_CFC_ (* Continuous Function Chart, elements in execution order *)
#0 OR(SCHU_P2_4_Z_M1_AV, NOT SCHU_P2_4_SA1_DI5_A)
#1 RT_Pusk:R_TRIG(CLK: SCHU_P2_4_UST_RE_PUSK)
#2 TON_PCH_OTKL:TON(IN: SCHU_P2_4_UST_RE_STOP, PT: T#1s)
#3 FT_PCH_OTKL:R_TRIG(CLK: #2.Q)
#4 RS_YA1_Open:RS(SET: #1.Q, RESET1: #3.Q)
#5 ZADERJ_SHOD_YA1:TON(IN: #4.Q1, PT: t#10s)
#6 TON_YA1_Z_ZAM_TE2:TON(IN: SCHU_P2_4_TE2_M_ZASCH, PT: t#5s)
#7 AND(#0, #21)
#8 AND(NOT SCHU_P2_4_SA1_DI5_A, NOT SCHU_P2_4_SA8_DI3_A, NOT SCHU_P2_4_SA1_DI6_M, NOT SCHU_P2_4_SA8_DI4_M)
#9 OR(#7, #8)
#10 TON_OTK_MV:TON(IN: #9, PT: t#5s)
#11 OR(#6.Q, Z_ZAM_SR, #10.Q)
#12 SEL(SCHU_P2_4_SA7_DI1_A, eHVAC2PointActuatorMode_Close_OP, eHVAC2PointActuatorMode_Auto_BMS)
#13 SEL(#11, #12, eHVAC2PointActuatorMode_Close_OP)
#14 fb_HVACPA:FB_HVAC2PointActuator(eHVACDataSecurityType_Idle, FALSE, TRUE, #5.Q, #13, SCHU_P2_4_KV1_DI4, SCHU_P2_4_YA1_DI6_ZKR, SCHU_P2_4_YA1_DI7_OTK, TRUE, SCHU_P2_4_SB, enableLimitSwitch, stokeTime)
#15 SCHU_P2_4_SA7_DO7_OTK <= #14.out 1
#16 OR(#14.out 4, #14.out 5)
#17 YA1_OTKAZ <= #16
#18 INT_TO_TIME(SCHU_P2_4_YA1_VREMYA_HODA)
#19 MUL(#18, 1000)
#20 stokeTime <= #19
#21 OR(SCHU_P2_4_Z_M2_AV, NOT SCHU_P2_4_SA8_DI3_A)
_END_CFC_
END_PROGRAM

(* POU IM/YA2_Upr, CFC *)
PROGRAM YA2_Upr
VAR
	YA2_PID: FB_HVACPIDCtrl;

	deadRange: REAL := 0.1;
	direction: BOOL;
	tTi: TIME;
	tTv: TIME;
	tTd: TIME;

	rYMin: REAL := 0;
	rYMax: REAL := 100;
	TON_SCHU_P2_4_P1_DI4_RUN: TON;
	reg1: BOOL;
	reg2: BOOL;

	SCHU_P2_4_YA2_: BOOL;
	YA2_REG_POL: BOOL;
	rwx: REAL;
	EPS1: REAL;
	EPS2: REAL;
END_VAR
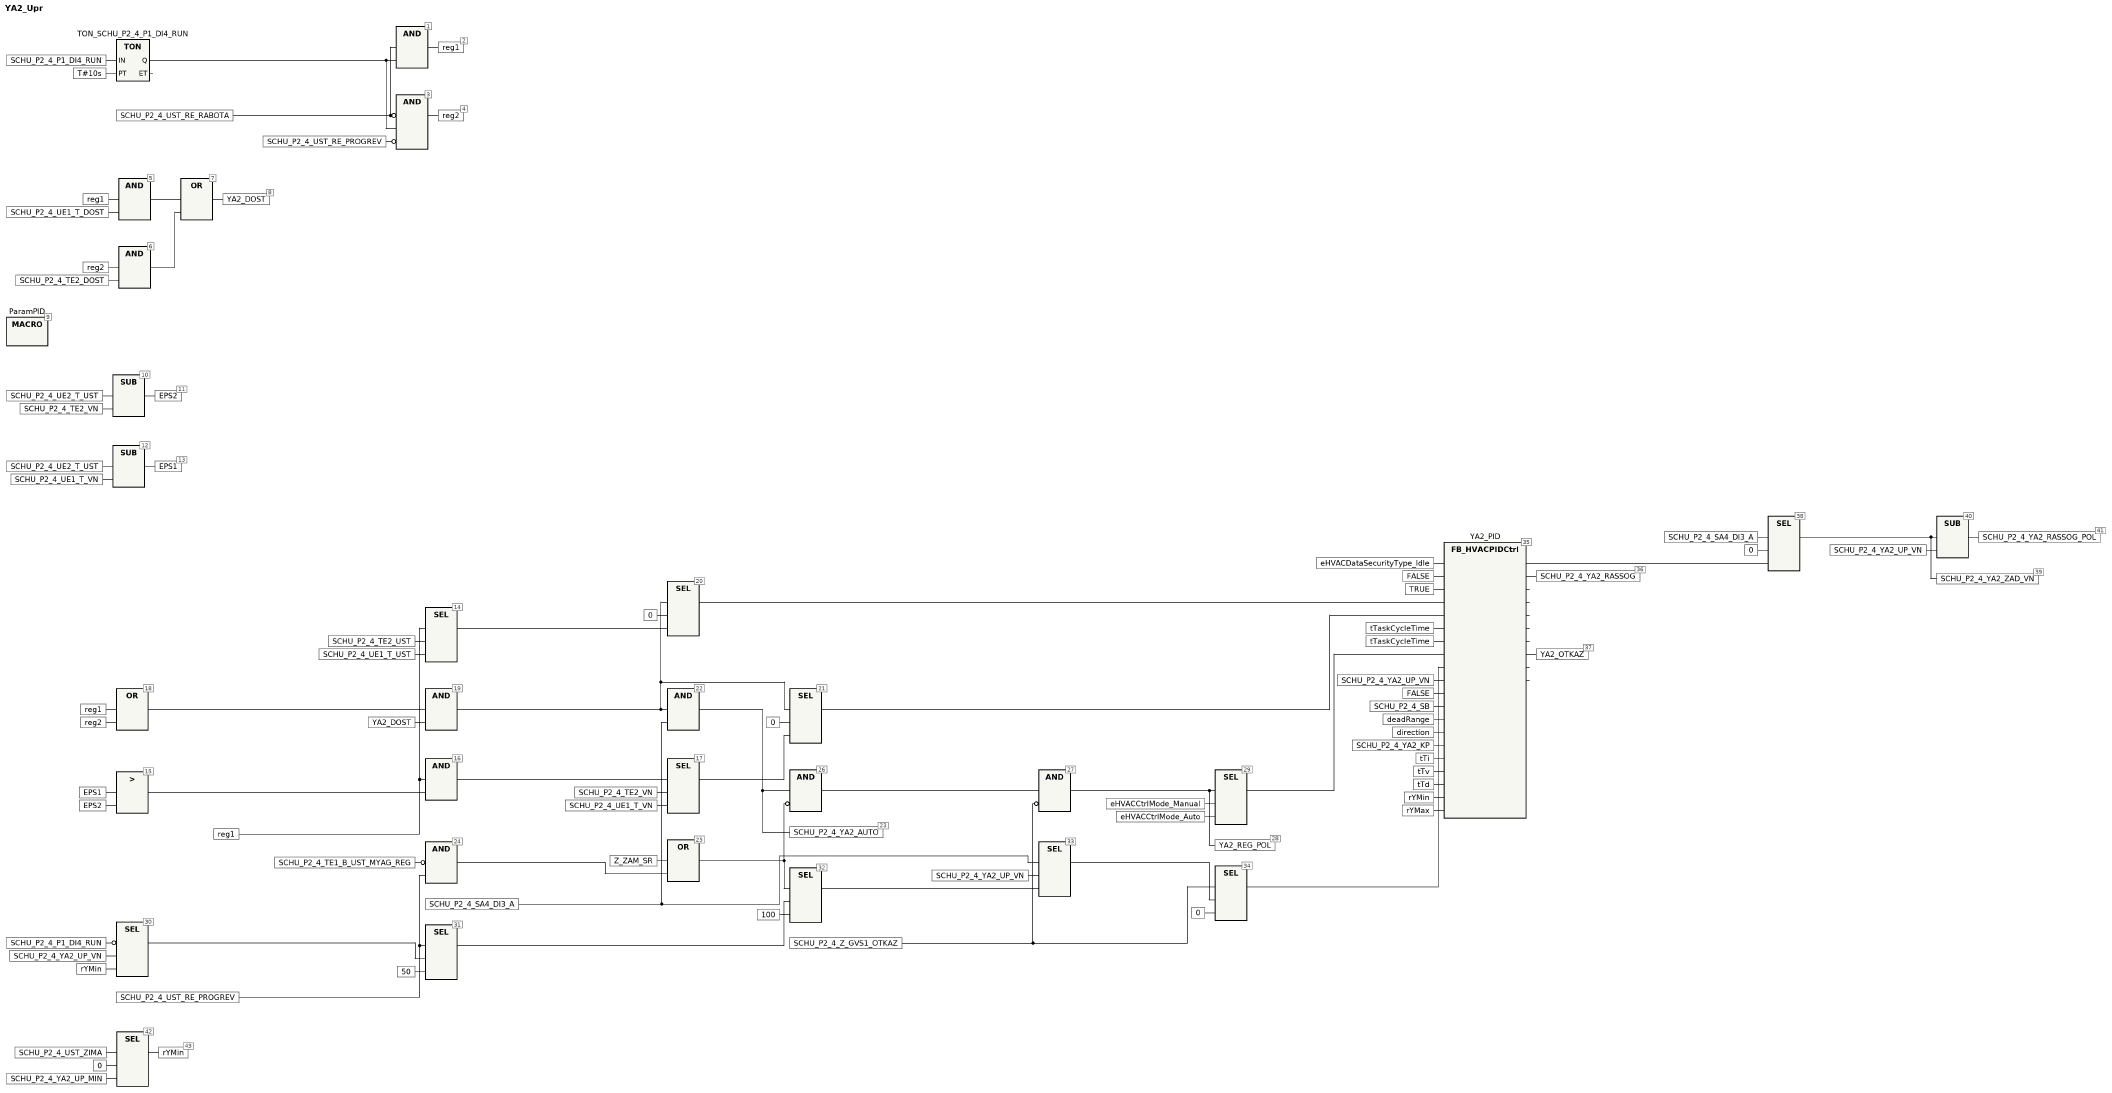
